RoboDK station: Yoavs_Hand_Simplified_UP6.rdk

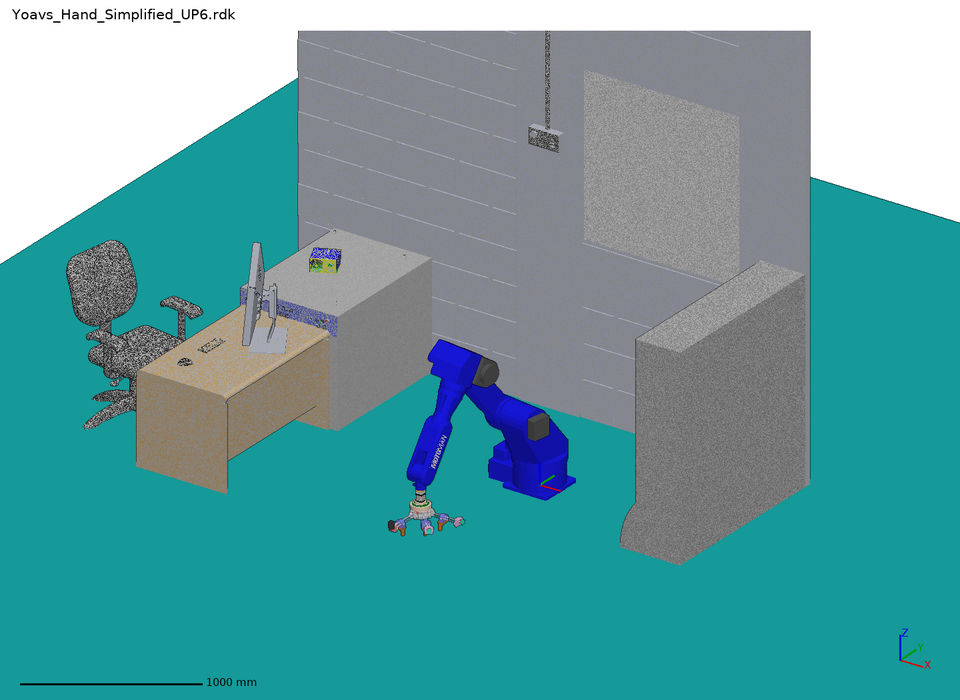
[picture v0: the station drawn from its stored meshes, robots at their saved joint values, targets as dots, program paths as lines]
Station Yoavs_Hand_Simplified_UP6. Poses are relative to the parent item; angles as X-Y-Z fixed-axis rotations.
  - frame Motoman UP6 Base at (0, 0, 0) mm
    - robot Motoman UP6: 6 axes, payload 6 kg, reach 1373 mm, repeatability 0.08 mm, weight 130 kg
        modified DH rows (alpha deg, a mm, theta deg, d mm): 0, 0, 0, 450; -90, 150, -90, 0; 0, 570, 0, 0; -90, 130, 0, 640; 90, 0, 90, 0; -90, 0, 0, 95
        joint limits [-170, -90, -170, -1, -135, -360] to [170, 155, 190, 1, 180, 360]; home [0, 0, 0, 0, 0, 0]; saved at [-98.196, 39.677, -19.593, 0, 59.27, -81.804]
      - tool Hand, TCP at (0, 0, 210) mm, rotated rx -180 ry 0 rz -180 deg, size 120 x 345.7 x 151.9 mm, geometry from Hand_Only.IGS
        - object Fingertip_0 at (0, 15.5, 0) mm, size 48 x 45 x 103.5 mm, geometry from Fingertip_Only.IGS
        - object Finger_2 at (0, 0, 0) mm, rotated rx 0 ry 0 rz 90 deg, size 56.5 x 258 x 48.5 mm, geometry from Finger_Only.IGS
        - object Fingertip_2 at (-55.5, 0, 0) mm, rotated rx 0 ry 0 rz 90 deg, size 48 x 45 x 103.5 mm, geometry from Fingertip_Only.IGS
        - object Finger_3 at (0, 0, 0) mm, rotated rx 0 ry 0 rz 45 deg, size 56.5 x 258 x 48.5 mm, geometry from Finger_Only.IGS
        - object Fingertip_3 at (-32.17, 32.17, 0) mm, rotated rx 0 ry 0 rz 45 deg, size 48 x 45 x 103.5 mm, geometry from Fingertip_Only.IGS
        - object Finger_1 at (0, 0, 0) mm, rotated rx 0 ry 0 rz 45 deg, size 56.5 x 258 x 48.5 mm, geometry from Finger_Only.IGS
        - object Fingertip_1 at (-32.17, 32.17, 0) mm, rotated rx 0 ry 0 rz 45 deg, size 48 x 45 x 103.5 mm, geometry from Fingertip_Only.IGS
  - Python program Hand_Control (listed below)
  - object Plane 4m x 4m at (0, 0, 0) mm, size 8000 x 8000 x 4 mm, geometry from plane_1m.sld
  - object Cardboard box at (-630, 300, 0) mm, rotated rx 0 ry 0 rz 45 deg, size 547.2 x 663.1 x 349.1 mm, geometry from Cardboard box.STEP
  - object Table Assembly at (-1350, -350, 760) mm, rotated rx 90 ry 0 rz -90 deg, size 1250 x 771 x 500 mm, geometry from Table Assembly.STEP
  - object Bookcase at (1180, -670, 750) mm, rotated rx -90 ry 0 rz 90 deg, size 2500 x 1500 x 350 mm, geometry from Bookcase.STEP
  - object Wall at (0, 910, 1500) mm, rotated rx 90 ry 0 rz 0 deg, size 4000 x 3000 x 100 mm, geometry from Wall.STEP
  - object Room Assembly at (-1020, 358, -190) mm, rotated rx 90 ry 0 rz -90 deg, size 1945 x 4060 x 3887.6 mm, geometry from Room Assembly.STEP

--- Python program Hand_Control ---
# This program allows moving gripper fingers
import sys # allows getting the passed argument parameters
from robodk import *

fingertip_offset = 115.5
fingertip_0_min = 0
fingertip_0_max = 144
fingertip_min = 0
fingertip_max = 131

if len(sys.argv) < 2:
    #print('Invalid parameters. This function must be called as MoveGripper(Gripper_Id, Distance)')
    #print('Number of arguments: ' + str(len(sys.argv)))
    #raise Exception('Invalid parameters provided: ' + str(sys.argv))
    entry = mbox('Lead Fingertip Distance', entry='0')
    entry2 = mbox('Finger 1 angle', entry = '45')
    entry3 = mbox('1st Fingertip Distance', entry='0')
    entry4 = mbox('Finger 2 angle', entry = '90')
    entry5 = mbox('2nd Fingertip Distance', entry='0')
    entry6 = mbox('Finger 3 angle, enter 0 if there \nare only two fingers and a thumb', entry = '135')
    entry7 = mbox('3rd Fingertip Distance', entry='0')
    if not entry:
        raise Exception('Operation cancelled by user')

    FINGERTIP_DISTANCE_0 = float(entry)
    FINGER_ANGLE_1 = float(entry2)
    FINGERTIP_DISTANCE_1 = float(entry3)
    FINGER_ANGLE_2 = float(entry4)
    FINGERTIP_DISTANCE_2 = float(entry5)
    FINGER_ANGLE_3 = float(entry6)
    FINGERTIP_DISTANCE_3 = float(entry7)

else:
    FINGERTIP_DISTANCE_0 = float(sys.argv[1])
    FINGER_ANGLE_1 = float(sys.argv[2])
    FINGERTIP_DISTANCE_1 = float(sys.argv[3])
    FINGER_ANGLE_2 = float(sys.argv[4])
    FINGERTIP_DISTANCE_2 = float(sys.argv[5])

    if len(sys.argv) < 6: #Three fingers
        FINGER_ANGLE_3 = 0
        FINGERTIP_DISTANCE_3 = 0
    else:
        FINGER_ANGLE_3 = float(sys.argv[6])
        FINGERTIP_DISTANCE_3 = float(sys.argv[7])


from robolink import *    # API to communicate with RoboDK
RDK = Robolink()

#Constants


fingertip_0 = RDK.Item('Fingertip_0')
fingertip_1 = RDK.Item('Fingertip_1')
finger_1 = RDK.Item('Finger_1')
fingertip_2 = RDK.Item('Fingertip_2')
finger_2 = RDK.Item('Finger_2')
fingertip_3 = RDK.Item('Fingertip_3')
finger_3 = RDK.Item('Finger_3')

if not fingertip_0.Valid():
    raise Exception('Invalid fingertip ID')

fingertip_0.setPose(transl(0,fingertip_offset-FINGERTIP_DISTANCE_0,0))

finger_1.setPose(rotz(FINGER_ANGLE_1*pi/180))
fingertip_1.setPose(rotz(FINGER_ANGLE_1*pi/180)*transl(0,fingertip_offset-FINGERTIP_DISTANCE_1,0))

finger_2.setPose(rotz(FINGER_ANGLE_2*pi/180))
fingertip_2.setPose(rotz(FINGER_ANGLE_2*pi/180)*transl(0,fingertip_offset-FINGERTIP_DISTANCE_2,0))

#Three Digit Hand case
if FINGER_ANGLE_3==0:
    FINGER_ANGLE_3 = FINGER_ANGLE_1
    FINGERTIP_DISTANCE_3=FINGERTIP_DISTANCE_1
    finger_3.setVisible(False)
    fingertip_3.setVisible(False)
else:
    finger_3.setVisible(True)
    fingertip_3.setVisible(True)


finger_3.setPose(rotz(FINGER_ANGLE_3*pi/180))
fingertip_3.setPose(rotz(FINGER_ANGLE_3*pi/180)*transl(0,fingertip_offset-FINGERTIP_DISTANCE_3,0))



# Set the station parameter
#RDK.setParam('Gripper', GRIPPER_VALUE)
